// TIA Portal V17 export
// export: Created 2024-09-02T12:50:04.6278132Z, ExportSetting WithDefaults, DisplayName Totally Integrated Automation Portal, DisplayVersion V17, DisplayName TIA Portal Openness, DisplayVersion V17, DisplayName TIA Portal Version Control Interface, DisplayVersion V17, DisplayName STEP 7 Professional, DisplayVersion V17, DisplayName STEP 7 Safety, DisplayVersion V17, DisplayName WinCC Professional, DisplayVersion V17
FUNCTION "AnwFC_Management_SQ" : Void   // FC1180, LAD
TITLE = Step sequence management / Schrittkettenverwaltung
{ S7_Optimized_Access := 'TRUE' }
AUTHOR : VAF
FAMILY : SK
NAME : SK
VERSION : 0.1
// stored: AutoNumber true, IsIECCheckEnabled false, SetENOAutomatically false, UDAEnableTagReadback false
   VAR_TEMP
      Motion_Release : Bool;   // Bewegungsfreigabe / Motion permit
      Hand : Bool;
      Auto : Bool;
   END_VAR
BEGIN

REGION Network 1: Motion permit - OP70 / Bewegungsfreigabe
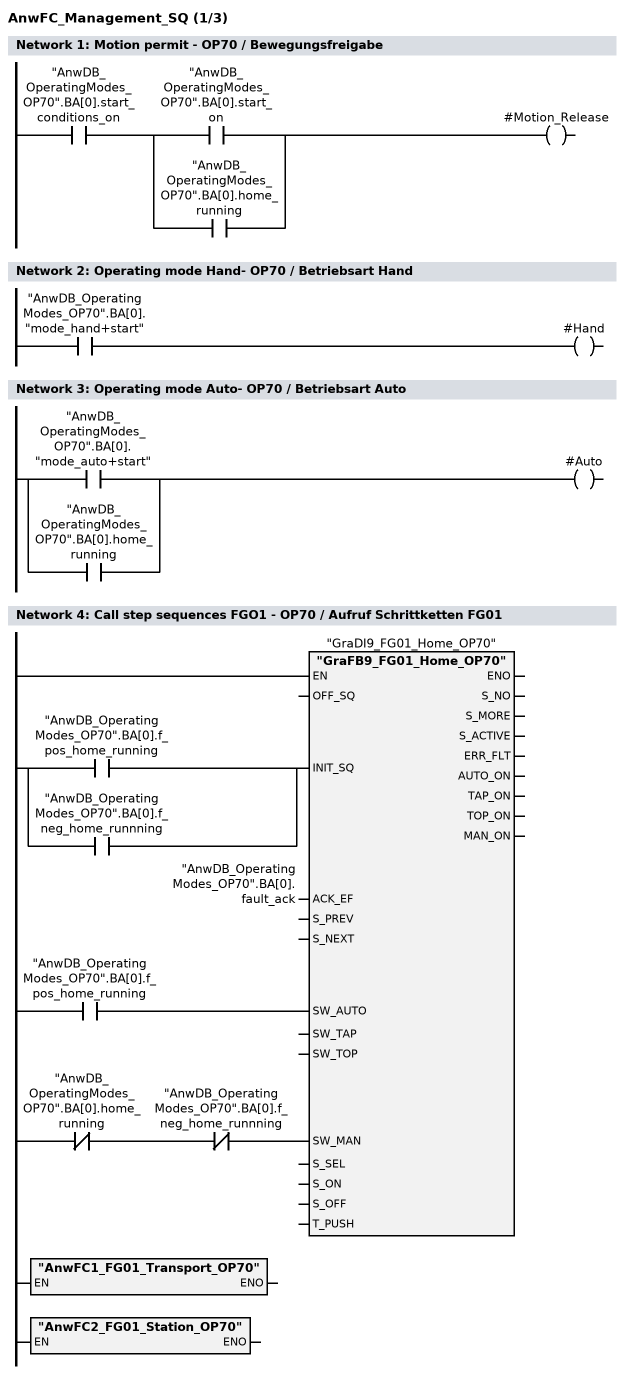
   RUNG wire#powerrail
      Contact( "AnwDB_OperatingModes_OP70".BA[0].start_conditions_on )
      wire#w1
      Contact( "AnwDB_OperatingModes_OP70".BA[0].start_on )
      wire#w2
      Coil( #Motion_Release )
   END_RUNG
   RUNG wire#w1
      Contact( "AnwDB_OperatingModes_OP70".BA[0].home_running )
   END_RUNG wire#w2
   // the same network as SCL:
   #Motion_Release := "AnwDB_OperatingModes_OP70".BA[0].start_conditions_on AND ("AnwDB_OperatingModes_OP70".BA[0].start_on OR "AnwDB_OperatingModes_OP70".BA[0].home_running);
END_REGION

REGION Network 2: Operating mode Hand- OP70 / Betriebsart Hand
   RUNG wire#powerrail
      Contact( "AnwDB_OperatingModes_OP70".BA[0]."mode_hand+start" )
      Coil( #Hand )
   END_RUNG
   // the same network as SCL:
   #Hand := "AnwDB_OperatingModes_OP70".BA[0]."mode_hand+start";
END_REGION

REGION Network 3: Operating mode Auto- OP70 / Betriebsart Auto
   RUNG wire#powerrail
      Contact( "AnwDB_OperatingModes_OP70".BA[0]."mode_auto+start" )
      wire#w1
      Coil( #Auto )
   END_RUNG
   RUNG wire#powerrail
      Contact( "AnwDB_OperatingModes_OP70".BA[0].home_running )
   END_RUNG wire#w1
   // the same network as SCL:
   #Auto := "AnwDB_OperatingModes_OP70".BA[0]."mode_auto+start" OR "AnwDB_OperatingModes_OP70".BA[0].home_running;
END_REGION

REGION Network 4: Call step sequences FGO1 - OP70 / Aufruf Schrittketten FG01
   RUNG wire#powerrail
      "GraDI9_FG01_Home_OP70"(INIT_SQ := wire#w1, SW_AUTO := wire#w2, SW_MAN := wire#w3, OFF_SQ :=, ACK_EF := "AnwDB_OperatingModes_OP70".BA[0].fault_ack, S_PREV :=, S_NEXT :=, SW_TAP :=, SW_TOP :=, S_SEL :=, S_ON :=, S_OFF :=, T_PUSH :=, S_NO =>, S_MORE =>, S_ACTIVE =>, ERR_FLT =>, AUTO_ON =>, TAP_ON =>, TOP_ON =>, MAN_ON =>)
   END_RUNG
   RUNG wire#powerrail
      Contact( "AnwDB_OperatingModes_OP70".BA[0].f_pos_home_running )
   END_RUNG wire#w1
   RUNG wire#powerrail
      Contact( "AnwDB_OperatingModes_OP70".BA[0].f_neg_home_runnning )
   END_RUNG wire#w1
   RUNG wire#powerrail
      Contact( "AnwDB_OperatingModes_OP70".BA[0].f_pos_home_running )
   END_RUNG wire#w2
   RUNG wire#powerrail
      I_Contact( "AnwDB_OperatingModes_OP70".BA[0].home_running )
      I_Contact( "AnwDB_OperatingModes_OP70".BA[0].f_neg_home_runnning )
   END_RUNG wire#w3
   RUNG wire#powerrail
      "AnwFC1_FG01_Transport_OP70"()
   END_RUNG
   RUNG wire#powerrail
      "AnwFC2_FG01_Station_OP70"()
   END_RUNG
   // the same network as SCL:
   "GraDI9_FG01_Home_OP70"(INIT_SQ := "AnwDB_OperatingModes_OP70".BA[0].f_pos_home_running OR "AnwDB_OperatingModes_OP70".BA[0].f_neg_home_runnning,   // "GraFB9_FG01_Home_OP70"
                           ACK_EF := "AnwDB_OperatingModes_OP70".BA[0].fault_ack,
                           SW_AUTO := "AnwDB_OperatingModes_OP70".BA[0].f_pos_home_running,
                           SW_MAN := NOT "AnwDB_OperatingModes_OP70".BA[0].home_running AND NOT "AnwDB_OperatingModes_OP70".BA[0].f_neg_home_runnning);
   "AnwFC1_FG01_Transport_OP70"();
   "AnwFC2_FG01_Station_OP70"();
END_REGION

REGION Network 5: Call step sequences FG02 - OP70 / Aufruf Schrittketten FG02
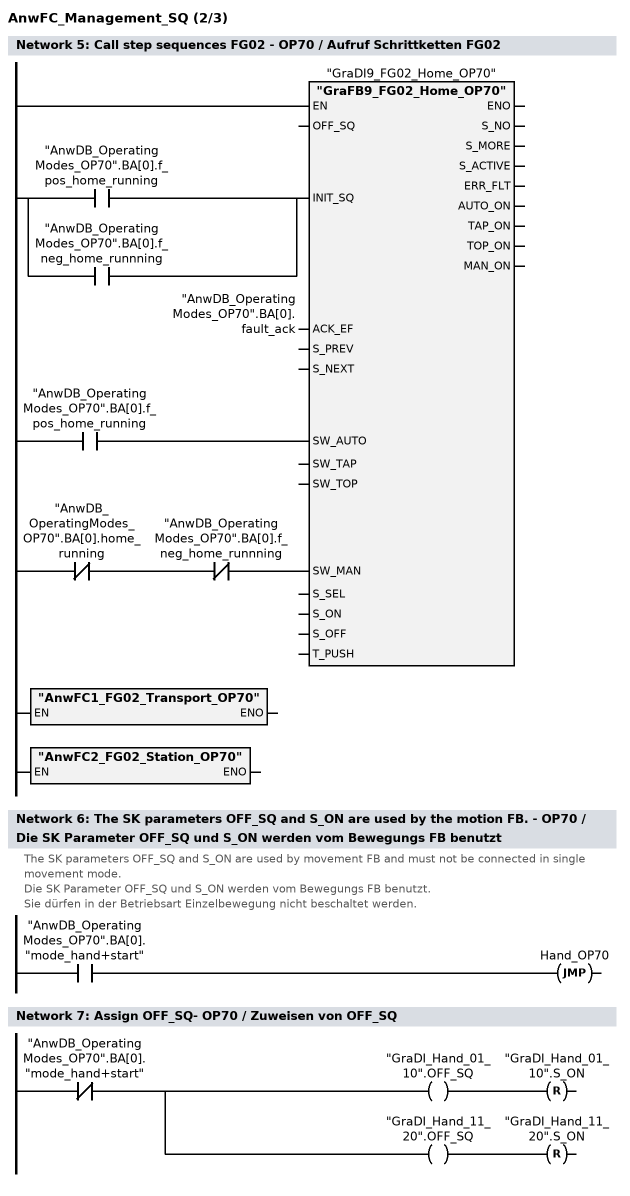
   RUNG wire#powerrail
      "GraDI9_FG02_Home_OP70"(INIT_SQ := wire#w1, SW_AUTO := wire#w2, SW_MAN := wire#w3, OFF_SQ :=, ACK_EF := "AnwDB_OperatingModes_OP70".BA[0].fault_ack, S_PREV :=, S_NEXT :=, SW_TAP :=, SW_TOP :=, S_SEL :=, S_ON :=, S_OFF :=, T_PUSH :=, S_NO =>, S_MORE =>, S_ACTIVE =>, ERR_FLT =>, AUTO_ON =>, TAP_ON =>, TOP_ON =>, MAN_ON =>)
   END_RUNG
   RUNG wire#powerrail
      Contact( "AnwDB_OperatingModes_OP70".BA[0].f_pos_home_running )
   END_RUNG wire#w1
   RUNG wire#powerrail
      Contact( "AnwDB_OperatingModes_OP70".BA[0].f_neg_home_runnning )
   END_RUNG wire#w1
   RUNG wire#powerrail
      Contact( "AnwDB_OperatingModes_OP70".BA[0].f_pos_home_running )
   END_RUNG wire#w2
   RUNG wire#powerrail
      I_Contact( "AnwDB_OperatingModes_OP70".BA[0].home_running )
      I_Contact( "AnwDB_OperatingModes_OP70".BA[0].f_neg_home_runnning )
   END_RUNG wire#w3
   RUNG wire#powerrail
      "AnwFC1_FG02_Transport_OP70"()
   END_RUNG
   RUNG wire#powerrail
      "AnwFC2_FG02_Station_OP70"()
   END_RUNG
   // the same network as SCL:
   "GraDI9_FG02_Home_OP70"(INIT_SQ := "AnwDB_OperatingModes_OP70".BA[0].f_pos_home_running OR "AnwDB_OperatingModes_OP70".BA[0].f_neg_home_runnning,   // "GraFB9_FG02_Home_OP70"
                           ACK_EF := "AnwDB_OperatingModes_OP70".BA[0].fault_ack,
                           SW_AUTO := "AnwDB_OperatingModes_OP70".BA[0].f_pos_home_running,
                           SW_MAN := NOT "AnwDB_OperatingModes_OP70".BA[0].home_running AND NOT "AnwDB_OperatingModes_OP70".BA[0].f_neg_home_runnning);
   "AnwFC1_FG02_Transport_OP70"();
   "AnwFC2_FG02_Station_OP70"();
END_REGION

REGION Network 6: The SK parameters OFF_SQ and S_ON are used by the motion FB. - OP70 / Die SK Parameter OFF_SQ und S_ON werden vom Bewegungs FB benutzt
   // The SK parameters OFF_SQ and S_ON are used by movement FB and must not be connected in single movement mode.
   // Die SK Parameter OFF_SQ und S_ON werden vom Bewegungs FB benutzt.
   // Sie dürfen in der Betriebsart Einzelbewegung nicht beschaltet werden.
   RUNG wire#powerrail
      Contact( "AnwDB_OperatingModes_OP70".BA[0]."mode_hand+start" )
      JumpCoil( Hand_OP70 )
   END_RUNG
   // the same network as SCL:
   IF "AnwDB_OperatingModes_OP70".BA[0]."mode_hand+start" THEN GOTO Hand_OP70; END_IF;
END_REGION

REGION Network 7: Assign OFF_SQ- OP70 / Zuweisen von OFF_SQ
   RUNG wire#powerrail
      I_Contact( "AnwDB_OperatingModes_OP70".BA[0]."mode_hand+start" )
      wire#w1
      Coil( "GraDI_Hand_01_10".OFF_SQ )
      R_Coil( "GraDI_Hand_01_10".S_ON )
   END_RUNG
   RUNG wire#w1
      Coil( "GraDI_Hand_11_20".OFF_SQ )
      R_Coil( "GraDI_Hand_11_20".S_ON )
   END_RUNG
   // the same network as SCL:
   "GraDI_Hand_01_10".OFF_SQ := NOT "AnwDB_OperatingModes_OP70".BA[0]."mode_hand+start";
   IF NOT "AnwDB_OperatingModes_OP70".BA[0]."mode_hand+start" THEN "GraDI_Hand_01_10".S_ON := FALSE; END_IF;
   "GraDI_Hand_11_20".OFF_SQ := NOT "AnwDB_OperatingModes_OP70".BA[0]."mode_hand+start";
   IF NOT "AnwDB_OperatingModes_OP70".BA[0]."mode_hand+start" THEN "GraDI_Hand_11_20".S_ON := FALSE; END_IF;
END_REGION

REGION Network 8: Calling the step chain manual (part 1/6)- OP70 / Aufruf der Schrittkette Hand (Teil 1/6)
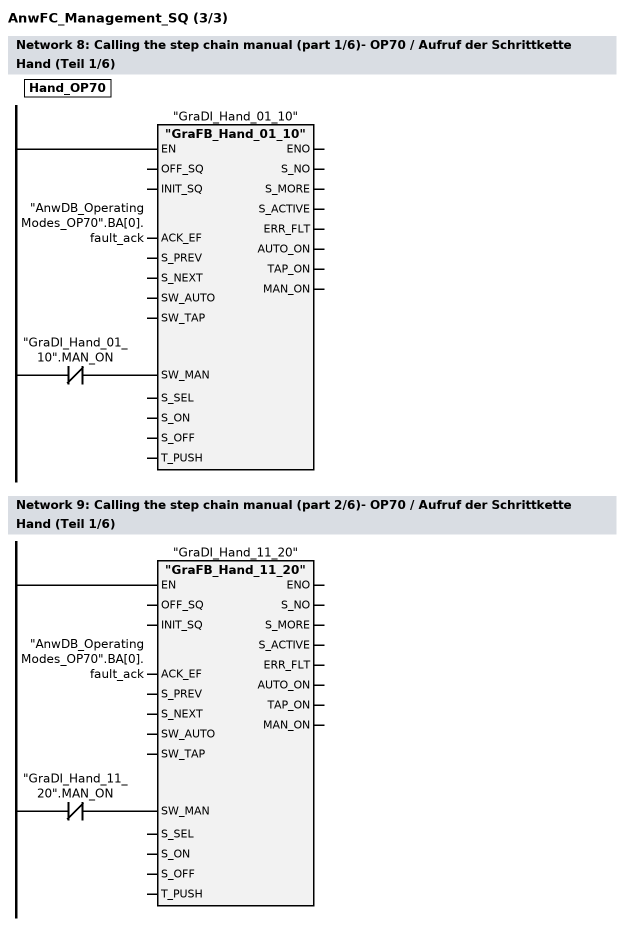
   Label( Hand_OP70 )
   RUNG wire#powerrail
      "GraDI_Hand_01_10"(SW_MAN := wire#w1, OFF_SQ :=, INIT_SQ :=, ACK_EF := "AnwDB_OperatingModes_OP70".BA[0].fault_ack, S_PREV :=, S_NEXT :=, SW_AUTO :=, SW_TAP :=, S_SEL :=, S_ON :=, S_OFF :=, T_PUSH :=, S_NO =>, S_MORE =>, S_ACTIVE =>, ERR_FLT =>, AUTO_ON =>, TAP_ON =>, MAN_ON =>)
   END_RUNG
   RUNG wire#powerrail
      I_Contact( "GraDI_Hand_01_10".MAN_ON )
   END_RUNG wire#w1
   // the same network as SCL:
   Hand_OP70:
   "GraDI_Hand_01_10"(ACK_EF := "AnwDB_OperatingModes_OP70".BA[0].fault_ack,   // "GraFB_Hand_01_10"
                      SW_MAN := NOT "GraDI_Hand_01_10".MAN_ON);
END_REGION

REGION Network 9: Calling the step chain manual (part 2/6)- OP70 / Aufruf der Schrittkette Hand (Teil 1/6)
   RUNG wire#powerrail
      "GraDI_Hand_11_20"(SW_MAN := wire#w1, OFF_SQ :=, INIT_SQ :=, ACK_EF := "AnwDB_OperatingModes_OP70".BA[0].fault_ack, S_PREV :=, S_NEXT :=, SW_AUTO :=, SW_TAP :=, S_SEL :=, S_ON :=, S_OFF :=, T_PUSH :=, S_NO =>, S_MORE =>, S_ACTIVE =>, ERR_FLT =>, AUTO_ON =>, TAP_ON =>, MAN_ON =>)
   END_RUNG
   RUNG wire#powerrail
      I_Contact( "GraDI_Hand_11_20".MAN_ON )
   END_RUNG wire#w1
   // the same network as SCL:
   "GraDI_Hand_11_20"(ACK_EF := "AnwDB_OperatingModes_OP70".BA[0].fault_ack,   // "GraFB_Hand_11_20"
                      SW_MAN := NOT "GraDI_Hand_11_20".MAN_ON);
END_REGION
END_FUNCTION
